Staubli VAL3: MotionPage.pgx

program MotionPage()
begin
  cls()
  bExit=false
  do
    call RefreshPage()
    call RefreshBelt()
    delay(0)
  until bExit
  bExit=false
end
